Fanuc KAREL source: kt00329.KL

-- PROVISIONAL review KL for V1013-1; original PC SHA256 b5e836bc60e6898978503f33e8dcb152c8a945da34032efbea1733723cb50f63
-- Incomplete behavior may be omitted. Consult companion uncertainty JSON. Do not deploy.
PROGRAM KT00329
%NOLOCKGROUP
VAR
  I1 : INTEGER
  I2 : INTEGER
  OUT : BOOLEAN
BEGIN
  -- UNRESOLVED_PC offsets 5-16; opcodes 2E,23
  -- UNRESOLVED_PC offsets 21-32; opcodes 2E,23
  -- UNRESOLVED_PC offsets 37-48; opcodes 2E,23
  -- UNRESOLVED_PC offsets 53-64; opcodes 2E,23
  -- UNRESOLVED_PC offsets 69-88; opcodes 21,21,59,23
  -- UNRESOLVED_PC offsets 93-97; opcodes 7F
END KT00329
